TEXTLIST TL_E_MESSAGETYPE
  0 = 'eMessageEmpty'
  1 = 'eMessageError'
  2 = 'eMessageWarning'
  3 = 'eMessageInfo'
  4 = 'eMessageVerbose'
   = ''
END_TEXTLIST

(* stored: Version 1.1.0.1, ProductVersion 3.1.4026.18
   TextList TL_E_MESSAGETYPE: Id {ea98c4cb-d547-44b8-b94a-d6667804ba0d} *)
